(* PLC project Beremiz Python Support Tests, LOLITECH Beremiz 0.0 *)
(* stored: creationDateTime 2008-12-14T16:21:19, modificationDateTime 2009-08-14T16:13:40 *)

PROGRAM main_pytest
  VAR
    counter : INT;
    DigitalBit0 : BOOL;
    DigitalBit1 : BOOL;
    DigitalBit2 : BOOL;
    DigitalBit3 : BOOL;
    DigitalBit4 : BOOL;
    DigitalBit5 : BOOL;
    DigitalBit6 : BOOL;
    DigitalBit7 : BOOL;
    Btn1 : Button;
    Btn2 : Button;
    Btn3 : Button;
    Btn4 : Button;
    Btn5 : Button;
    Btn6 : Button;
    Btn7 : Button;
    Btn8 : Button;
    Start_Stop : Button;
    Compteur : TextCtrl;
    Temoin : Led;
  END_VAR
  VAR  (* added by the conversion: wires and edge detectors of the diagram *)
    _AND96_OUT : BOOL;
    _ADD32_ENO : BOOL;
    _ADD32_OUT : INT;
  END_VAR

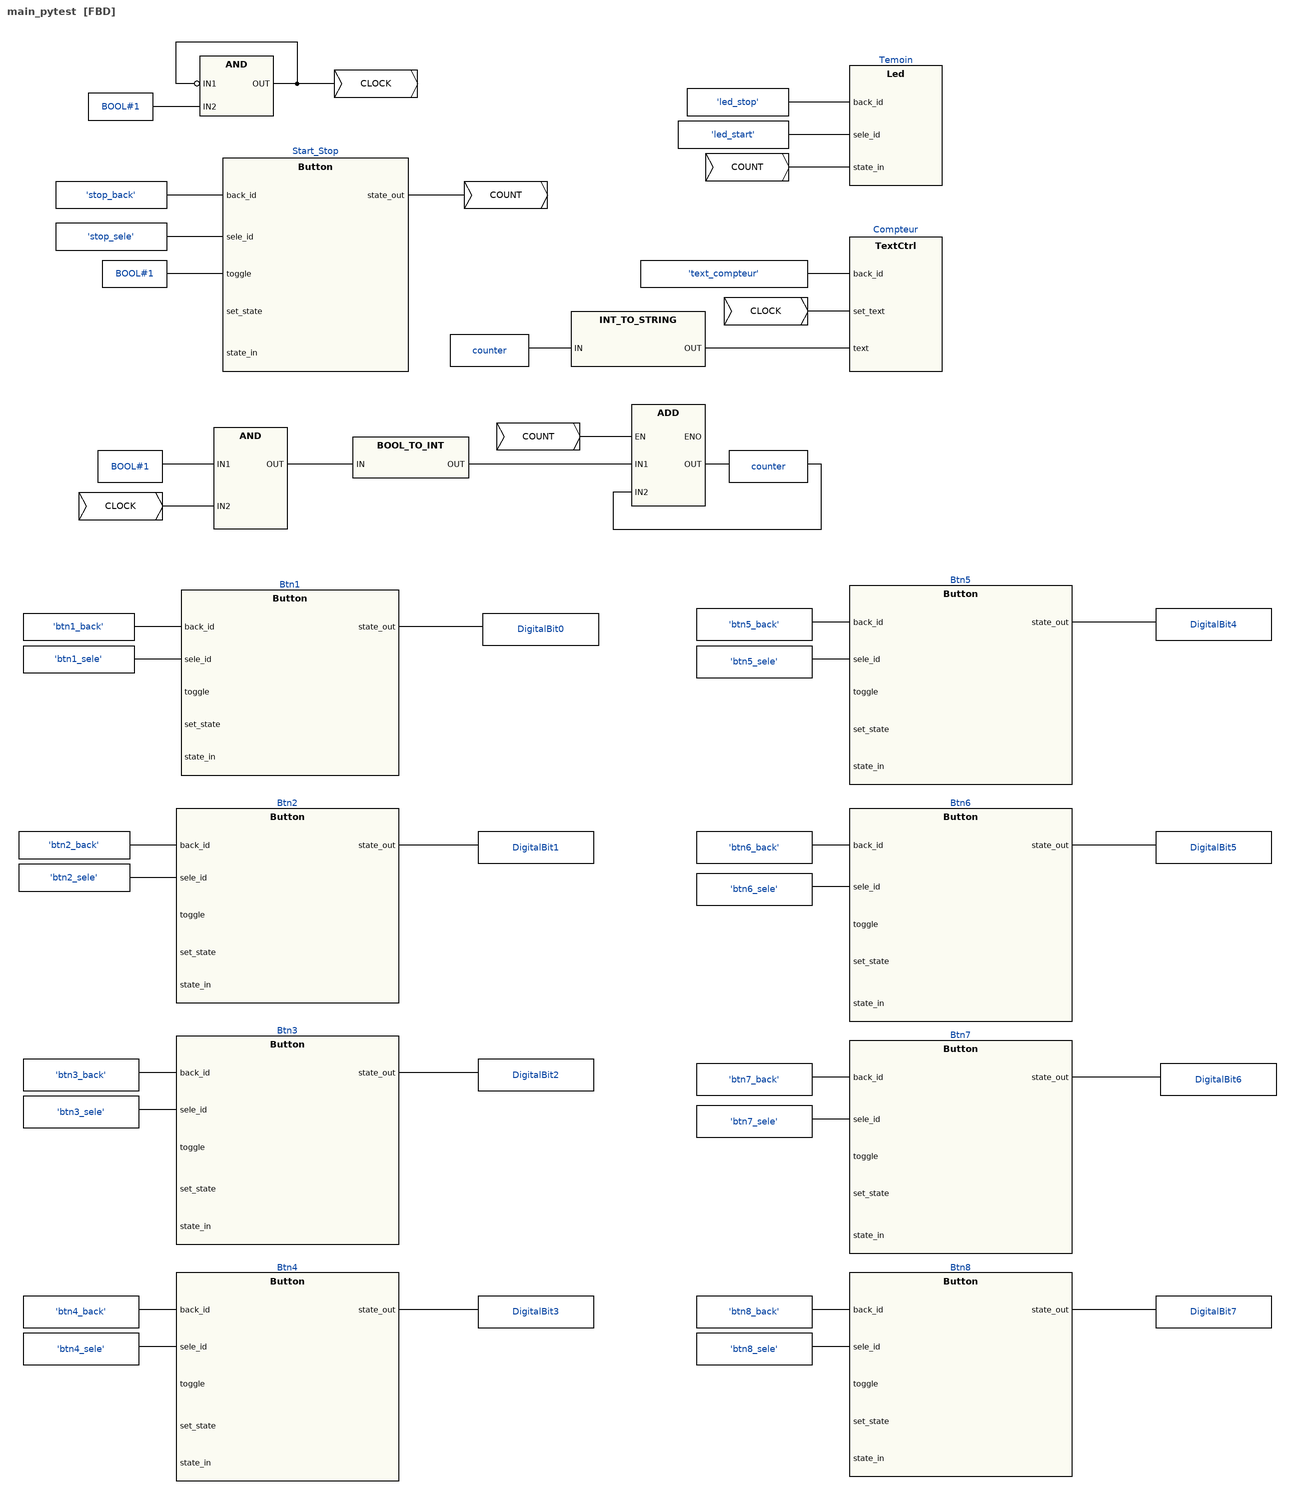
(* FBD diagram, written out as Structured Text *)
Start_Stop(back_id := 'stop_back', sele_id := 'stop_sele', toggle := BOOL#1);
_AND96_OUT := NOT _AND96_OUT AND BOOL#1;
_ADD32_OUT := ADD(EN := Start_Stop.state_out, IN1 := BOOL_TO_INT(BOOL#1 AND _AND96_OUT), IN2 := counter, ENO => _ADD32_ENO);
IF _ADD32_ENO THEN counter := _ADD32_OUT; END_IF;
Btn1(back_id := 'btn1_back', sele_id := 'btn1_sele');
DigitalBit0 := Btn1.state_out;
Btn5(back_id := 'btn5_back', sele_id := 'btn5_sele');
DigitalBit4 := Btn5.state_out;
Btn2(back_id := 'btn2_back', sele_id := 'btn2_sele');
DigitalBit1 := Btn2.state_out;
Btn6(back_id := 'btn6_back', sele_id := 'btn6_sele');
DigitalBit5 := Btn6.state_out;
Btn3(back_id := 'btn3_back', sele_id := 'btn3_sele');
DigitalBit2 := Btn3.state_out;
Btn7(back_id := 'btn7_back', sele_id := 'btn7_sele');
DigitalBit6 := Btn7.state_out;
Btn4(back_id := 'btn4_back', sele_id := 'btn4_sele');
DigitalBit3 := Btn4.state_out;
Btn8(back_id := 'btn8_back', sele_id := 'btn8_sele');
DigitalBit7 := Btn8.state_out;
Temoin(back_id := 'led_stop', sele_id := 'led_start', state_in := Start_Stop.state_out);
Compteur(back_id := 'text_compteur', set_text := _AND96_OUT, text := INT_TO_STRING(counter));
END_PROGRAM

CONFIGURATION conf_pytest
  RESOURCE res_pytest ON PLC
    TASK pytest_task(INTERVAL := t#100ms, PRIORITY := 0);
    PROGRAM pytest_instance : main_pytest;
  END_RESOURCE
END_CONFIGURATION
